Universal Robots PolyScope program: bearing_orient_from_upsidedown.urp

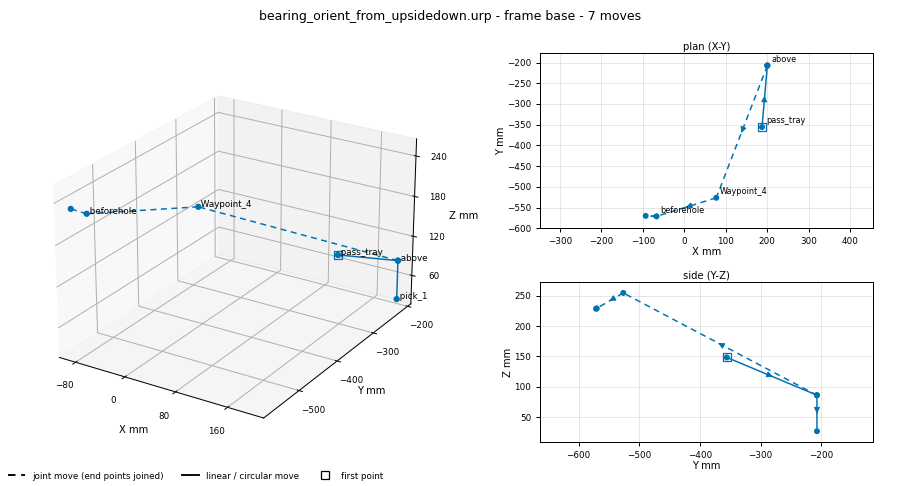
[picture p0: tool path of bearing_orient_from_upsidedown.urp in frame base, 7 of 11 moves have a stored position in this frame; points joined in program order, loops and branches not executed]
Program bearing_orient_from_upsidedown (installation=default directory=/programs/wrs2020 createdIn=5.7.0.90932 lastSavedIn=5.10.0.106288 robotSerialNumber=20205500607)
Calibrated DH parameters: a=[0.000096, -0.337, -0.383372, 0.000118, 0.000015, 0]; d=[0.162724, 79.377998, -95.545185, 16.300583, 0.099689, 0.099499]; alpha=[1.569249, 0.003272, 0.005201, 1.570041, -1.570219, 0]; deltaTheta=[0, 0.65664, 5.410619, 0.215927, -0.000001, 0]
Robot Program (runOnlyOnce=true)
  SuppressedNode
    MoveJ speed 60 deg/s, acceleration 80 deg/s^2 (useActiveTCP=true) feature=Base
      URCap Gripper (Robotiq_Grippers, Robotiq Inc.) dataModel(position=0.0, force=0.0, speed=100.0, positionInDouble=0.0, forceInDouble=0.0, speedInDouble=100.0, slaveIds=[9], blocking=true)
      Waypoint above_grasp: TCP in base x=151.464 y=-541.697 z=141.179 mm, rx=0.0942 ry=-3.1024 rz=0.0162 rad; joints [93.096, -77.216, 103.232, -116.53, -91.83, -0.395] deg; TCP offset x=0 y=0 z=165 mm, rx=0 ry=0 rz=0 rad
      Waypoint at_grasp: TCP in base x=151.456 y=-541.711 z=44.649 mm, rx=0.0942 ry=-3.1024 rz=0.0163 rad; joints [93.069, -69.788, 109.936, -130.663, -91.843, -0.332] deg
      URCap Gripper (Robotiq_Grippers, Robotiq Inc.) dataModel(position=100.0, force=100.0, speed=100.0, positionInDouble=100.0, forceInDouble=100.0, speedInDouble=100.0, slaveIds=[9], blocking=true)
  currentpose := get_actual_joint_positions()
  MoveJ speed 60 deg/s, acceleration 80 deg/s^2 (useActiveTCP=true) feature=Base
    Waypoint Waypoint (Variable): variable(name=currentpose)
    Waypoint pass_tray: TCP in base x=187.718 y=-355.766 z=148.266 mm, rx=0.1175 ry=3.1177 rz=-0.0239 rad; joints [97.948, -100.949, 126.425, -116.523, -88.651, 12.221] deg
  SuppressedNode
    Folder Center grasp and turn over
      MoveL speed 600 mm/s, acceleration 1200 mm/s^2 (useActiveTCP=true) feature=Base
        Waypoint pass_tray: TCP in base x=187.718 y=-355.766 z=148.266 mm, rx=0.1175 ry=3.1177 rz=-0.0239 rad; joints [97.948, -100.949, 126.425, -116.523, -88.651, 12.221] deg
        Waypoint above: motionParameters(blendRadius=0.05); TCP in base x=200.55 y=-207.27 z=86.012 mm, rx=0.028 ry=3.1154 rz=0.0066 rad; joints [105.259, -116.491, 145.894, -119.54, -88.262, 16.238] deg
        Waypoint pick_1: TCP in base x=200.551 y=-207.243 z=26.686 mm, rx=1.7859 ry=2.5612 rz=0.0285 rad; joints [105.196, -107.078, 152.162, -135.219, -88.267, 85] deg
      URCap Gripper (Robotiq_Grippers, Robotiq Inc.) dataModel(position=14.901960784313726, force=0.0, speed=0.0, positionInDouble=14.901960784313726, forceInDouble=0.0, speedInDouble=0.0, slaveIds=[9], blocking=true)
      MoveL speed 600 mm/s, acceleration 1200 mm/s^2 (useActiveTCP=true) feature=Base
        Waypoint turn_left (Relative): relativeFromPosition TCP in base x=217.155 y=-247.662 z=15.637 mm, rx=1.248 ry=2.8551 rz=-0.0099 rad; joints [106.781, -96.81, 148.171, -142.561, -88.879, 64.086] deg; TCP in base x=217.136 y=-247.633 z=15.614 mm, rx=-1.1429 ry=2.9115 rz=-0.0354 rad; joints [106.78, -96.81, 148.175, -142.562, -88.881, -26] deg
      URCap Gripper (Robotiq_Grippers, Robotiq Inc.) dataModel(position=100.0, force=0.0, speed=0.0, positionInDouble=100.0, forceInDouble=0.0, speedInDouble=0.0, slaveIds=[9], blocking=true)
      URCap Gripper (Robotiq_Grippers, Robotiq Inc.) dataModel(position=16.470588235294116, force=100.0, speed=100.0, positionInDouble=16.470588235294116, forceInDouble=100.0, speedInDouble=100.0, slaveIds=[9], blocking=true)
      MoveL speed 600 mm/s, acceleration 1200 mm/s^2 (useActiveTCP=true) feature=Base
        Waypoint turn_left (Relative): relativeFromPosition TCP in base x=217.155 y=-247.662 z=15.637 mm, rx=1.248 ry=2.8551 rz=-0.0099 rad; joints [106.781, -96.81, 148.171, -142.561, -88.879, 64.086] deg; TCP in base x=217.136 y=-247.633 z=15.614 mm, rx=-1.1429 ry=2.9115 rz=-0.0354 rad; joints [106.78, -96.81, 148.175, -142.562, -88.881, -26] deg
        SuppressedNode
          Waypoint incline (Relative): relativeFromPosition TCP in base x=218.308 y=-500.893 z=48.171 mm, rx=-2.1842 ry=2.228 rz=-0.0241 rad; joints [98.786, -72.218, 112.617, -130.37, -88.156, -79.999] deg; TCP in base x=222.438 y=-500.865 z=43.608 mm, rx=-1.9097 ry=1.9461 rz=-0.5 rad; joints [85.345, -72.496, 119.917, -134.528, -60.233, -94.253] deg
        Waypoint very_inclined: TCP in base x=204.089 y=-207.342 z=29.992 mm, rx=-1.8382 ry=1.2743 rz=-0.6818 rad; joints [61.986, -91.809, 150.898, -100.204, -56.445, -154.149] deg
      URCap Gripper (Robotiq_Grippers, Robotiq Inc.) dataModel(position=100.0, force=100.0, speed=100.0, positionInDouble=100.0, forceInDouble=100.0, speedInDouble=100.0, slaveIds=[9], blocking=true)
  SuppressedNode
    Folder Turn over
      MoveL speed 250 mm/s, acceleration 1200 mm/s^2 (useActiveTCP=true) feature=Base
        Waypoint Waypoint_1: TCP in base x=204.646 y=-207.137 z=60.413 mm, rx=-2.2092 ry=1.5298 rz=-0.3992 rad; joints [78.452, -115.617, 150.776, -108.098, -65.239, -125.981] deg
        Waypoint Waypoint_2: TCP in base x=204.647 y=-207.117 z=60.401 mm, rx=2.0312 ry=-1.4027 rz=-0.5577 rad; joints [139.677, -86.614, 134.601, -113.442, -126.285, -52.88] deg
        Waypoint Waypoint_3: TCP in base x=204.642 y=-207.147 z=27.003 mm, rx=2.0311 ry=-1.4028 rz=-0.5576 rad; joints [139.655, -81.582, 136.497, -120.357, -126.29, -52.849] deg
        URCap Gripper (Robotiq_Grippers, Robotiq Inc.) dataModel(position=16.470588235294116, force=100.0, speed=100.0, positionInDouble=16.470588235294116, forceInDouble=100.0, speedInDouble=100.0, slaveIds=[9], blocking=true)
        Waypoint Waypoint_5: TCP in base x=200.941 y=-208.521 z=28.795 mm, rx=-1.71 ry=1.186 rz=-0.7602 rad; joints [58.642, -82.323, 148.613, -96.034, -55.779, -162.097] deg
        URCap Gripper (Robotiq_Grippers, Robotiq Inc.) dataModel(position=100.0, force=100.0, speed=100.0, positionInDouble=100.0, forceInDouble=100.0, speedInDouble=100.0, slaveIds=[9], blocking=true)
        Waypoint Waypoint_6: motionParameters(blendRadius=0); TCP in base x=216.054 y=-236.414 z=98.791 mm, rx=-1.655 ry=2.0482 rz=-0.194 rad; joints [82.397, -112.212, 142.807, -104.225, -64.36, -89.314] deg
  Folder Center grasp and pick inclined
    MoveL speed 600 mm/s, acceleration 1200 mm/s^2 (useActiveTCP=true) feature=Base
      SuppressedNode
        Waypoint pass_tray: TCP in base x=187.718 y=-355.766 z=148.266 mm, rx=0.1175 ry=3.1177 rz=-0.0239 rad; joints [97.948, -100.949, 126.425, -116.523, -88.651, 12.221] deg
      Waypoint above: motionParameters(blendRadius=0.034); TCP in base x=200.55 y=-207.27 z=86.012 mm, rx=0.028 ry=3.1154 rz=0.0066 rad; joints [105.259, -116.491, 145.894, -119.54, -88.262, 16.238] deg
      Waypoint pick_1: TCP in base x=200.551 y=-207.243 z=26.686 mm, rx=1.7859 ry=2.5612 rz=0.0285 rad; joints [105.196, -107.078, 152.162, -135.219, -88.267, 85] deg
    URCap Gripper (Robotiq_Grippers, Robotiq Inc.) dataModel(position=15.0, force=100.0, speed=100.0, positionInDouble=15.0, forceInDouble=100.0, speedInDouble=100.0, slaveIds=[9], blocking=true)
    MoveL speed 600 mm/s, acceleration 1200 mm/s^2 (useActiveTCP=true) feature=Base
      Waypoint turn_left (Relative): relativeFromPosition TCP in base x=217.155 y=-247.662 z=15.637 mm, rx=1.248 ry=2.8551 rz=-0.0099 rad; joints [106.781, -96.81, 148.171, -142.561, -88.879, 64.086] deg; TCP in base x=217.136 y=-247.633 z=15.614 mm, rx=-1.1429 ry=2.9115 rz=-0.0354 rad; joints [106.78, -96.81, 148.175, -142.562, -88.881, -26] deg
      SuppressedNode
        Waypoint turn_right (Relative): relativeFromPosition TCP in base x=217.14 y=-247.643 z=15.618 mm, rx=-1.143 ry=2.9115 rz=-0.0354 rad; joints [106.781, -96.809, 148.175, -142.565, -88.882, -26.001] deg; TCP in base x=217.147 y=-247.646 z=15.617 mm, rx=1.2481 ry=2.8551 rz=-0.0099 rad; joints [106.78, -96.808, 148.173, -142.561, -88.879, 64.088] deg
    URCap Gripper (Robotiq_Grippers, Robotiq Inc.) dataModel(position=100.0, force=0.0, speed=0.0, positionInDouble=100.0, forceInDouble=0.0, speedInDouble=0.0, slaveIds=[9], blocking=true)
    URCap Gripper (Robotiq_Grippers, Robotiq Inc.) dataModel(position=16.470588235294116, force=100.0, speed=100.0, positionInDouble=16.470588235294116, forceInDouble=100.0, speedInDouble=100.0, slaveIds=[9], blocking=true)
    MoveL speed 600 mm/s, acceleration 1200 mm/s^2 (useActiveTCP=true) feature=Base
      SuppressedNode
        Waypoint pick_1: TCP in base x=200.551 y=-207.243 z=26.686 mm, rx=1.7859 ry=2.5612 rz=0.0285 rad; joints [105.196, -107.078, 152.162, -135.219, -88.267, 85] deg
      Waypoint turn_left (Relative): relativeFromPosition TCP in base x=217.155 y=-247.662 z=15.637 mm, rx=1.248 ry=2.8551 rz=-0.0099 rad; joints [106.781, -96.81, 148.171, -142.561, -88.879, 64.086] deg; TCP in base x=217.136 y=-247.633 z=15.614 mm, rx=-1.1429 ry=2.9115 rz=-0.0354 rad; joints [106.78, -96.81, 148.175, -142.562, -88.881, -26] deg
      Waypoint incline (Relative): relativeFromPosition TCP in base x=218.308 y=-500.893 z=48.171 mm, rx=-2.1842 ry=2.228 rz=-0.0241 rad; joints [98.786, -72.218, 112.617, -130.37, -88.156, -79.999] deg; TCP in base x=222.438 y=-500.865 z=43.608 mm, rx=-1.9097 ry=1.9461 rz=-0.5 rad; joints [85.345, -72.496, 119.917, -134.528, -60.233, -94.253] deg
    URCap Gripper (Robotiq_Grippers, Robotiq Inc.) dataModel(position=100.0, force=100.0, speed=100.0, positionInDouble=100.0, forceInDouble=100.0, speedInDouble=100.0, slaveIds=[9], blocking=true)
  MoveL speed 600 mm/s, acceleration 1200 mm/s^2 (useActiveTCP=false) tcp=gripper_85_tip; feature=Base
    Waypoint above: TCP in base x=200.55 y=-207.27 z=86.012 mm, rx=0.028 ry=3.1154 rz=0.0066 rad; joints [105.259, -116.491, 145.894, -119.54, -88.262, 16.238] deg
  MoveJ speed 180 deg/s, acceleration 360 deg/s^2 (useActiveTCP=false) tcp=gripper_85_tip; feature=Base
    Waypoint Waypoint_4: motionParameters(blendRadius=0.05); TCP in base x=77.346 y=-526.445 z=254.497 mm, rx=2.1138 ry=-1.9338 rz=-0.2706 rad; joints [93.109, -85.443, 98.102, -105.695, -107.975, -92.542] deg
    Waypoint beforehole: TCP in base x=-66.725 y=-571.237 z=228.439 mm, rx=1.497 ry=-1.6176 rz=-0.8285 rad; joints [93.116, -71.584, 102.92, -120.139, -149.991, -81.706] deg
    Waypoint athole: TCP in base x=-93.062 y=-570.055 z=228.956 mm, rx=1.497 ry=-1.6176 rz=-0.8285 rad; joints [90.445, -71.97, 104.758, -126.218, -149.936, -87.03] deg
